(* IEC 61131-3 sources: ae-json-library/test, 3 files *)

(* ---- TestMyProgram.st ---- *)
USING Simatic.Ax.Json;

NAMESPACE Simatic.Ax.UseJsonLibrary
    {TestFixture}
    CLASS TestMyProgram
    VAR
        timeOfOperations : LTIME;
        doc : JsonDocument;
        cmpBuff : ARRAY[0..20] OF CHAR;
        buffer : ARRAY[0..999] OF CHAR;
        myBoolean : JsonBoolean := (Value := TRUE, Key := 'myBoolean');
        myInt : JsonInt := (Value := 1234, Key := 'myInt');
        myDint : JsonDInt := (Value := DINT#12345678, Key := 'myDint');
        myObject : JsonObject := (Key := 'myObject');
        step : Steps;
        deserializer : Deserializer;
        key : STRING;
        keyFound : BOOL;
        intValue : INT;
    END_VAR
    {Test}
    METHOD PUBLIC MyTestMethod
        VAR_TEMP
            i : DINT;
        END_VAR

        FOR i := 1 TO 10000 DO
            this.MyProgram();
        END_FOR;

    END_METHOD

    METHOD PUBLIC MyProgram

        VAR_TEMP
            keyArray : ARRAY[0..1] OF STRING;
        END_VAR
        CASE step OF
            Steps#CreateDocument1:
                // Create Document 1st object model
                // Expected Value: {"myInt": 1234}
                doc.AddElement(myInt);
                doc.Serialize();
                step := Steps#SerializeDocument1
                ;
            Steps#SerializeDocument1:
                // Serialize Document 1st object model1
                doc.Serialize();
                step := Steps#ParseDocument1
                ;
            Steps#ParseDocument1:
                // Parse Document 1st object model
                deserializer.buffer := REF(buffer);
                key := 'myInt';
                keyFound := deserializer.TryParse(key, intValue);
                step := Steps#ResetJSonDocument1
                ;
            Steps#ResetJSonDocument1:
                // ResetJSonDocument 1st object model
                doc.Reset();
                step := Steps#CreateDocument2
                ;
            Steps#CreateDocument2:
                // Create Document 2nd object model (nested object)
                // Expected Value: {"myBoolean": true, "myObject": {"myInt": 1234, "myDint": 12345678}}
                myObject.AddElement(myInt);
                myObject.AddElement(myDint);
                doc.AddElement(myBoolean);
                doc.AddElement(myObject);
                step := Steps#SerializeDocument2
                ;
            Steps#SerializeDocument2:
                // Serialize Document 2nd object model including time meassurement
                doc.Serialize();
                step := Steps#ParseDocument2;
                ;
            Steps#ParseDocument2:
                // Parse Document 1st object model
                // Get Values from a nested element
                deserializer.buffer := REF(buffer);
                keyArray[0] := 'myObject';
                keyArray[1] := 'myInt';
                keyFound := deserializer.TryParse(keyArray, intValue);
                step := Steps#ResetJSonDocument2;
                ;
            Steps#ResetJSonDocument2:
                // ResetJSonDocument 2nd configuration
                doc.Reset();
                step := Steps#CreateDocument1;
                ;
        END_CASE;
    END_METHOD
    END_CLASS
END_NAMESPACE

(* ---- UsingDeserializer.st ---- *)
USING Simatic.Ax.Conversion;
USING AxUnit.Assert;
USING System.Strings;
USING Simatic.Ax.Json;

{TestFixture}
Class UsingDeserializer
    VAR protected
        deserializer : Deserializer;
        buffer : ARRAY[0..999] OF CHAR;

        JSON_Entry: STRING;
        key: STRING;
        len:DINT;
        keyFound: BOOL;

    END_VAR

    {Test}
    Method Public GetValue_BASIC_DATA_TYPES
        VAR
            stringValue: STRING;
            usintValue: USINT;
            intValue: INT;
        END_VAR

        //Getting JSON and convert it to ARRAY OF CHAR
        JSON_Entry := '{ "key1": "stringValue", "key2": 10, "key3": 1234, "key4": "1234"}';
        len:= Strings.ToArray.OfCharCount(str := JSON_Entry, arr := buffer);

        //Give it to the deserializer
        deserializer.SetBuffer(REF(buffer));

        //Parse string
        key:= 'key1';
        keyFound := deserializer.TryParse( key, stringValue);

        Equal(keyFound, TRUE);
        Equal(stringValue, 'stringValue');

        //Parse usint
        key:= 'key2';
        keyFound := deserializer.TryParse( key, usintValue);

        Equal(keyFound, TRUE);
        Equal(usintValue, usint#10);

        //Parse int
        key:= 'key3';
        keyFound := deserializer.TryParse( key, intValue);

        Equal(keyFound, TRUE);
        Equal(intValue, 1234);

        //FailedParsing
        key:= 'Not a key';
        keyFound := deserializer.TryParse( key, intValue);

        Equal(keyFound, FALSE);
        Equal(intValue, 0);

        //Parse foreign datatypes int to string -> possible
        key:= 'key2';
        keyFound := deserializer.TryParse( key, stringValue);

        Equal(keyFound, TRUE);
        Equal(stringValue, '10');

        //Parse foreign datatypes string to int -> possible if string is a int
        key:= 'key4';
        keyFound := deserializer.TryParse( key, intValue);

        Equal(keyFound, TRUE);
        Equal(intValue, 1234);

         //Parse foreign datatypes string to int -> False if string is not a int
         key:= 'key1';
         keyFound := deserializer.TryParse( key, intValue);

         Equal(keyFound, FALSE);
         Equal(intValue, 0);
    END_Method

    {Test}
    Method Public GetValue_ARRAY
        VAR
            stringValue: STRING;
        END_VAR

        JSON_Entry := '{ "arraykey": [1234, 5678]}';

        len:= Strings.ToArray.OfCharCount(str := JSON_Entry, arr := buffer);
        deserializer.SetBuffer(REF(buffer));

        key:= 'arraykey';
        keyFound := deserializer.TryParse( key, stringValue);

        Equal(keyFound, TRUE);
        Equal(stringValue, '[1234, 5678]');
    END_Method

    {Test}
    Method Public GetValue_Nested
        VAR
            stringValue: STRING;
            keyArray: ARRAY[0..1] OF STRING;
        END_VAR

        JSON_Entry := '{ "key1": {"nestedkey1": "nested value", "nestedkey2": 456}}';

        len:= Strings.ToArray.OfCharCount(str := JSON_Entry, arr := buffer);
        deserializer.SetBuffer(REF(buffer));

        //Parse string
        key:= 'key1';
        keyFound := deserializer.TryParse( key, stringValue);

        Equal(keyFound, TRUE);
        Equal(stringValue, '{"nestedkey1": "nested value", "nestedkey2": 456}'); //right now there is a 254 character limit!

        //Get Values from a nested element
        keyArray[0] := 'key1';
        keyArray[1] := 'nestedkey1';

        keyFound := deserializer.TryParse( keyArray, stringValue);

        Equal(keyFound, TRUE);
        Equal(stringValue, 'nested value');
    END_Method

    {Test}
    Method Public GetValue_Nested_in_Nested
        VAR
            stringValue: STRING;
            keyArray: ARRAY[0..2] OF STRING;
            intValue: INT;
        END_VAR

        JSON_Entry := '{ "key1": {"nestedkey1": "nested value", "nestedkey2": {"nested_nested_key" : 1234}}}';

        len:= Strings.ToArray.OfCharCount(str := JSON_Entry, arr := buffer);
        deserializer.SetBuffer(REF(buffer));

        //Get Values from a nested element
        keyArray[0] := 'key1';
        keyArray[1] := 'nestedkey2';
        keyArray[2] := 'nested_nested_key';

        keyFound := deserializer.TryParse( keyArray, intValue);

        Equal(keyFound, TRUE);
        Equal(intValue, 1234);
    END_Method

END_CLASS

(* ---- UsingSerializer.st ---- *)
USING AxUnit.Assert;
USING System.Strings;
USING Simatic.Ax.Conversion;
USING Simatic.Ax.Json;

NAMESPACE Simatic.Ax.UseJsonLibrary
    {TestFixture}
    Class UsingSerializer
        VAR
            doc : JsonDocument;
            docStateLess : JsonDocument;
            cmpBuff : ARRAY[0..20] OF CHAR;
            buffer : ARRAY[0..999] OF CHAR;

            str, s : STRING;

            myBoolean : JsonBoolean := (Value := TRUE, Key := 'myBoolean');
            myInt : JsonInt := (Value := 1234, Key := 'myInt');
            myDint : JsonDInt := (Value := DINT#12345678, Key := 'myDint');
            myString : JsonString := (Value := 'this is my string', Key := 'myString');
            myObject : JsonObject := (Key := 'myObject');
        END_VAR

        // This method will be called before each test method
        {TestSetup}
        METHOD PUBLIC MyTestSetup
            doc := docStateLess;
        END_METHOD

        {Test}
        METHOD PUBLIC Serialize_BOOLEAN
            doc.AddElement(myBoolean);
            doc.buffer := REF(buffer);
            doc.buffer := REF(buffer);
            doc.buffer := REF(buffer);
            doc.Serialize();

            str := Arrays.ToString(buffer, 0, 18);
            //Equal(expected := '{"myBoolean": true}', actual := str);
        END_METHOD

        {Test}
        METHOD PUBLIC Serialize_INT
            doc.AddElement(myInt);
            doc.buffer := REF(buffer);
            doc.Serialize();

            str := Arrays.ToString(buffer, 0, 14);
            //Equal(expected := '{"myInt": 1234}', actual := str);
        END_METHOD

        {Test}
        METHOD PUBLIC Serialize_DINT
            doc.AddElement(myDint);
            doc.buffer := REF(buffer);
            doc.Serialize();

            str := Arrays.ToString(buffer, 0, 19);
            //Equal(expected := '{"myDint": 12345678}', actual := str);
        END_METHOD

        {Test}
        METHOD PUBLIC Serialize_STRING
            doc.AddElement(myString);
            doc.buffer := REF(buffer);
            doc.buffer := REF(buffer);
            doc.Serialize();

            str := Arrays.ToString(buffer, 0, 32);
            //Equal(expected := '{"myString": "this is my string"}', actual := str);
        END_METHOD

        {Test}
        METHOD PUBLIC Serialize_INT_DINT
            doc.AddElement(myInt);
            doc.AddElement(myDint);
            doc.buffer := REF(buffer);
            doc.buffer := REF(buffer);
            doc.buffer := REF(buffer);
            doc.Serialize();

            str := Arrays.ToString(buffer, 0, 34);
            //Equal(expected := '{"myInt": 1234, "myDint": 12345678}', actual := str);
        END_METHOD

        {Test}
        METHOD PUBLIC Serialize_and_reset_NestedObject
            myObject.AddElement(myInt);
            myObject.AddElement(myDint);

            doc.AddElement(myBoolean);
            doc.AddElement(myObject);
            doc.buffer := REF(buffer);
            doc.Serialize();

            str := Arrays.ToString(buffer, 0, 67);
            //Equal(expected := '{"myBoolean": true, "myObject": {"myInt": 1234, "myDint": 12345678}}', actual := str);

            // Reset document
            doc.Reset();

            // Create new document
            myObject.AddElement(myInt);
            myObject.AddElement(myDint);

            doc.AddElement(myBoolean);
            doc.AddElement(myObject);
            doc.buffer := REF(buffer);
            doc.buffer := REF(buffer);
            doc.Serialize();
            str := Arrays.ToString(buffer, 0, 67);
            //Equal(expected := '{"myBoolean": true, "myObject": {"myInt": 1234, "myDint": 12345678}}', actual := str);

        END_METHOD
    END_CLASS
END_NAMESPACE
